Staubli VAL3: checkAdvMoves.pgx

program checkAdvMoves()
  local num l_nIndex
begin

  //setMutex(bAdvMoves)
  for l_nIndex=0 to size(bAdvMoveBusy)-1
    if bAdvMoveBusy[l_nIndex]
      if taskStatus(sAdvMovePrefix+toString("",l_nIndex))==-1
        bAdvMoveBusy[l_nIndex]=false
      endIf
    endIf
  endFor
  //bAdvMoves=false

end
